KUKA KRL program: Program1.src, Program1.dat

--- Program1.src ---
&ACCESS RV
DEF Program1 ( )

END

--- Program1.dat ---
&ACCESS RV
DEFDAT Program1 PUBLIC

ENDDAT
